Universal Robots PolyScope program: 5.12.2024.urp

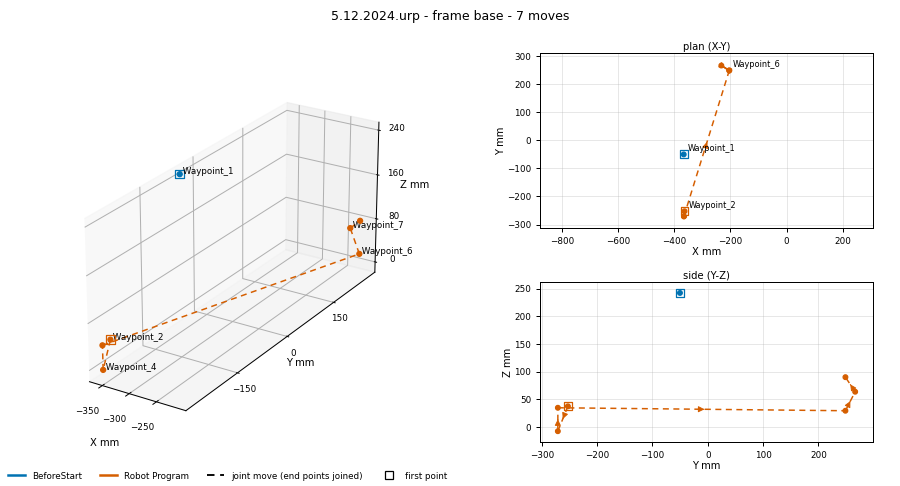
[picture p0: tool path of 5.12.2024.urp in frame base, 7 of 7 moves have a stored position in this frame; points joined in program order, loops and branches not executed]
Program 5.12.2024 (installation=default directory=/programs createdIn=3.15.8.106339 lastSavedIn=3.15.8.106339 robotSerialNumber=2023330214)
Calibrated DH parameters: a=[-0.000161, -0.243516, -0.175941, 0.000055, -0.000127, 0]; d=[0.151869, -0.926342, 57.568096, -56.529557, 0.085345, 0.082309]; alpha=[1.571543, -0.007517, 0.002128, 1.570286, -1.573097, 0]; deltaTheta=[0.000048, 0.028487, 0.571925, -0.600676, 0.000055, 0.000013]
BeforeStart
  MoveJ speed 60 deg/s, acceleration 80 deg/s^2 (useActiveTCP=true)
    Waypoint Waypoint_1: TCP in base x=-366.565 y=-50.19 z=242.41 mm, rx=-0.456 ry=-2.9947 rz=0.0702 rad; joints [-149.336, -89.622, -91.185, -82.431, 88.033, -2201.798] deg; flange x=-321.283 y=-59.011 z=320.94 mm, rx=-0.456 ry=-2.9947 rz=0.0702 rad
Robot Program (runOnlyOnce=false)
  MoveJ speed 60 deg/s, acceleration 80 deg/s^2 (useActiveTCP=true)
    Waypoint Waypoint_2: TCP in base x=-363.667 y=-252.721 z=37.531 mm, rx=0.1444 ry=-3.114 rz=0.0196 rad; joints [-126.819, -127.618, -95.209, -45.593, 89.201, -2201.802] deg; flange x=-324.383 y=-248.124 z=119.572 mm, rx=0.1444 ry=-3.114 rz=0.0196 rad
    Waypoint Waypoint_4: TCP in base x=-365.903 y=-270.898 z=-7.467 mm, rx=-0.4242 ry=3.1119 rz=-0.0107 rad; joints [-126.601, -137.107, -91.487, -41.017, 90.075, -2211.82] deg; flange x=-329.925 y=-260.311 z=75.532 mm, rx=-0.4242 ry=3.1119 rz=-0.0107 rad
    Waypoint Waypoint_5: TCP in base x=-365.911 y=-270.852 z=34.886 mm, rx=-0.424 ry=3.1119 rz=-0.0106 rad; joints [-126.604, -130.125, -90.246, -49.244, 90.115, -2211.798] deg; flange x=-329.933 y=-260.278 z=117.885 mm, rx=-0.424 ry=3.1119 rz=-0.0106 rad
    Waypoint Waypoint_6: TCP in base x=-204.329 y=248.851 z=29.521 mm, rx=-1.6481 ry=-2.6423 rz=0.003 rad; joints [-206.105, -108.71, -134.951, -24.617, 89.871, -2211.758] deg; flange x=-185.825 y=214.109 z=111.655 mm, rx=-1.6481 ry=-2.6423 rz=0.003 rad
    Waypoint Waypoint_7: TCP in base x=-232.574 y=266.465 z=63.846 mm, rx=-1.4046 ry=-2.1517 rz=-0.8373 rad; joints [-184.46, -120.14, -146.066, 2.737, 46.43, -2190.407] deg; flange x=-215.299 y=184.497 z=99.598 mm, rx=-1.4046 ry=-2.1517 rz=-0.8373 rad
    Waypoint Waypoint_8: TCP in base x=-204.366 y=248.867 z=90.178 mm, rx=-1.6481 ry=-2.6421 rz=0.0031 rad; joints [-206.116, -93.474, -128.685, -46.112, 90.003, -2211.785] deg; flange x=-185.855 y=214.124 z=172.31 mm, rx=-1.6481 ry=-2.6421 rz=0.0031 rad
